ABB RobotStudio station: Solution4.rspag

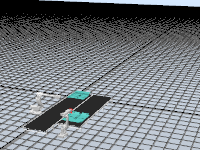
--- station ---
Station Solution4 (saved by RobotStudio 20.4.9280.0)
Controller Controlador1
  mechanical unit ROB_1: IRB6620_150_220__01, 6 joints, base frame (9000, 3450, 0) mm, rotated rx 0 ry 0 rz 180 deg
Layout (positions relative to the parent item):
  - Belt_IN1 [part]
  - IRB7600_150_350__03 [mechanism, from Robots\IRB7600_150_350_G_03.rslib] at (5500, -1300, 0) mm, rotated rx 0 ry 0 rz 90 deg; joint values [0, 0, 0, 0, 0.5236, 0] (rad or m)
  - IRB6620_150_220__01 [mechanism, from Robots\IRB6620_150_220_G_01.rslib] at (9000, 3450, 0) mm, rotated rx 0 ry 0 rz 180 deg; joint values [0, 0, 0, 0, 0.5236, 0] (rad or m)
  - Vacuum Tool [mechanism] at (7619.79, 3450, 1755) mm, rotated rx 180 ry 60 rz 0 deg
      TCP tVacuum at (0, 0, 200) mm
      links: Vacuum Tool
  - Belt Conveyor [part]
  - Carpet [part] at (1440.36, 1252.7, 780) mm, rotated rx 0 ry 0 rz 90 deg
  - Carpet_2 [part] at (6559.64, 3547.3, 780) mm, rotated rx 0 ry 0 rz -90 deg
Attachment: Vacuum Tool is attached to IRB6620_150_220__01 / Link6
Station signals: DI Positioner
Targets, tools, work objects and paths stored in the station and not in the controller backup, written as RAPID:
! task T_ROB1
MODULE CalibData
  PERS tooldata tVacuum:=[TRUE,[[0,0,200],[1,0,0,0]],[15,[0,0,133.333333333],[1,0,0,0],0,0,0]];
ENDMODULE


--- Backups/Controlador1/RAPID/TASK1/PROGMOD/Module1.mod ---
MODULE Module1
    !***********************************************************
    !
    ! Módulo:  Module1
    !
    ! Descripción:
    !   <Introduzca la descripción aquí>
    !
    ! Autor: Alex
    !
    ! Versión: 1.0
    !
    !***********************************************************


    !***********************************************************
    !
    ! Procedimiento Main
    !
    !   Este es el punto de entrada de su programa
    !
    !***********************************************************
    PROC main()
        !Añada aquí su código
    ENDPROC
ENDMODULE
